// Mitsubishi GX Works2 project: final project   PLC: Q03UDV

PROGRAM MAIN
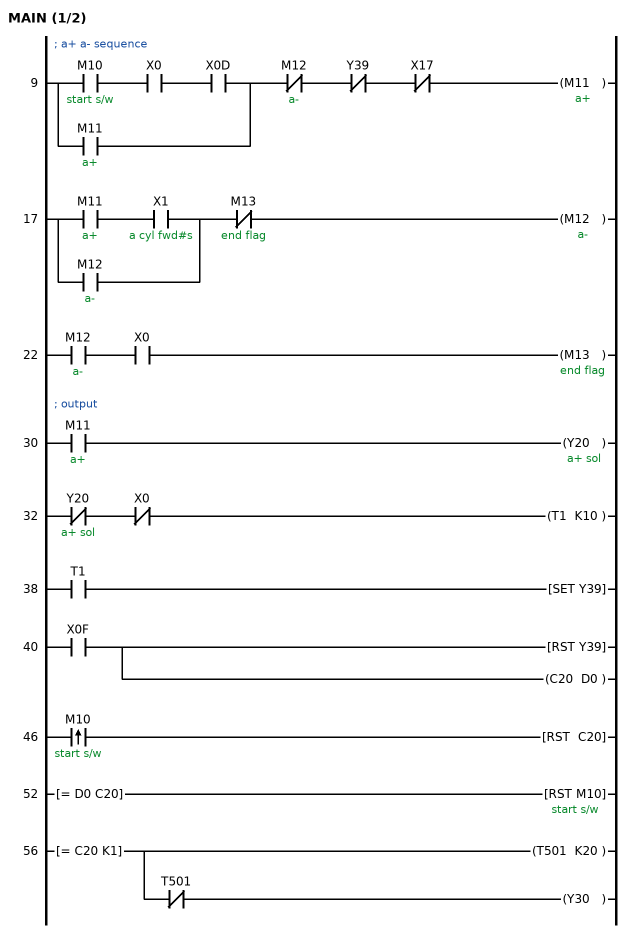
; a+ a- sequence
9     LD      M10  ; start s/w
      AND     X0
      AND     X0D
      OR      M11  ; a+
      ANI     M12  ; a-
      ANI     Y39
      ANI     X17
      OUT     M11  ; a+
17    LD      M11  ; a+
      AND     X1  ; a cyl fwd#s
      OR      M12  ; a-
      ANI     M13  ; end flag
      OUT     M12  ; a-
22    LD      M12  ; a-
      AND     X0
      OUT     M13  ; end flag
; output
30    LD      M11  ; a+
      OUT     Y20  ; a+ sol
32    LDI     Y20  ; a+ sol
      ANI     X0
      OUT     T1 K10
38    LD      T1
      SET     Y39
40    LD      X0F
      RST     Y39
      OUT     C20 D0
46    LDP     M10  ; start s/w
      RST     C20
52    LD=     D0 C20
      RST     M10  ; start s/w
56    LD=     C20 K1
      OUT     T501 K20
      ANI     T501
      OUT     Y30
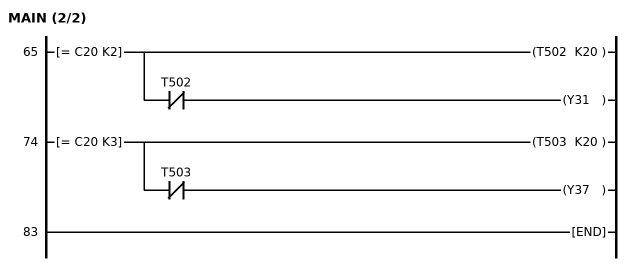
65    LD=     C20 K2
      OUT     T502 K20
      ANI     T502
      OUT     Y31
74    LD=     C20 K3
      OUT     T503 K20
      ANI     T503
      OUT     Y37
83    END
END_PROGRAM

// device comments not shown above
M1000  ; end flag
